// TwinCAT 3 PLC project MicroTestStandWFS
// ProgramVersion: 3.1.4020.5
// libraries:
//   lcls-twincat-motion, * (SLAC)
//   lcls2-cc-lib, * (SLAC)
//   PMPS, * (SLAC - LCLS)
//   Tc2_Standard, * (Beckhoff Automation GmbH)
//   Tc2_System, * (Beckhoff Automation GmbH)
//   Tc2_Utilities, * (Beckhoff Automation GmbH)
//   Tc3_Module, * (Beckhoff Automation GmbH)
//   VisuDialogs
//   VisuSymbols,3.5.10.0,System
// project tree:
//   DUTs/ DUT_MotionStage_Extras.TcDUT (not stored)
//   / GlobalTextList.TcGTLO, PlcTask.TcTTO (not stored), VISU_TASK.TcTTO (not stored)
//   POUs/ Main.TcPOU
//   VISUs/ Visualization.TcVIS, VisualizationManager.TcVMO (not stored), VISU_MotionStage.TcVIS (not stored)

// ---- POUs/Main.TcPOU
PROGRAM Main
VAR
	{attribute 'TcLinkTo' := '.bLimitForwardEnable  := TIIB[EL7041-Y]^STM Status^Status^Digital input 1;
	                          .bLimitBackwardEnable := TIIB[EL7041-Y]^STM Status^Status^Digital input 2;
	                          .bBrakeRelease        := TIIB[EL2004]^Channel 1^Output'}
	M1: DUT_MotionStage;
	M1_Extras: DUT_MotionStage_Extras;
    
	M2: DUT_MotionStage;
	M2_Extras: DUT_MotionStage_Extras;
	
	{attribute 'TcLinkTo' := '.fbThermoCouple1.bError := TIIB[EL3314]^TC Inputs Channel 1^Status^Error;
							  .fbThermoCouple1.bUnderrange := TIIB[EL3314]^TC Inputs Channel 1^Status^Underrange;
							  .fbThermoCouple1.bOverrange := TIIB[EL3314]^TC Inputs Channel 1^Status^Overrange;
							  .fbThermoCouple1.iRaw := TIIB[EL3314]^TC Inputs Channel 1^Value;
							  .fbThermoCouple2.bError := TIIB[EL3314]^TC Inputs Channel 2^Status^Error;
							  .fbThermoCouple2.bUnderrange := TIIB[EL3314]^TC Inputs Channel 2^Status^Underrange;
							  .fbThermoCouple2.bOverrange := TIIB[EL3314]^TC Inputs Channel 2^Status^Overrange;
							  .fbThermoCouple2.iRaw := TIIB[EL3314]^TC Inputs Channel 2^Value'}
	fbWFS: FB_WFS;
	

    {attribute 'TcLinkTo' := 'TIIB[EL5042]^FB Inputs Channel 2^Position'}
	iM1RawEncoder AT %I*: ULINT;
	iM1AdjustedEncoder: UDINT;
    
    {attribute 'TcLinkTo' := 'TIIB[EL5042]^FB Inputs Channel 1^Position'}
    iM2RawEncoder AT %I*: ULINT;
    iM2AdjustedEncoder: UDINT;
    
	iMaxLINT: ULINT := 18446744073709551615;
	
	bStartup: BOOL := TRUE;
    
    // PMPS Machinery
    fbArbiterIO: FB_SubSysToArbiter_IO;
    {attribute 'pytmc' := 'pv: PLC:TST:MOT:ARB'}
    fbArbiter: FB_Arbiter(1);
    {attribute 'pytmc' := 'pv: PLC:TST:MOT:FFO:01'}
    fbFFHWO: FB_HardwareFFOutput := (bAutoReset := TRUE);
END_VAR

fbWFS(
    stYStage := M1,
    stZStage := M2,
    fbArbiter := fbArbiter,
    fbFFHWO:=fbFFHWO);

fbFFHWO.Execute();
fbArbiterIO(
    Arbiter:=fbArbiter,
    fbFFHWO:=fbFFHWO);


iM1AdjustedEncoder := ULINT_TO_UDINT(iMaxLINT - iM1RawEncoder) + 1;
iM2AdjustedEncoder := ULINT_TO_UDINT(iM2RawEncoder);

M1_Extras.bVisuHighLim := NOT M1.bAllForwardEnable;
M1_Extras.bVisuLowLim := NOT M1.bAllBackwardEnable;
M2_Extras.bVisuHighLim := NOT M2.bAllForwardEnable;
M2_Extras.bVisuLowLim := NOT M2.bAllBackwardEnable;

IF bStartup THEN
	bStartup := FALSE;
	M1.fVelocity := 1;
	M1.fAcceleration := 200;
	M1.fDeceleration := 200;
	M2.fVelocity := 1;
	M2.fAcceleration := 200;
	M2.fDeceleration := 200;
END_IF

END_PROGRAM

// ---- GlobalTextList.TcGTLO
TEXTLIST GlobalTextList
  593 = '%f'
  964 = '%X'
  957 = '+'
  951 = '-'
  960 = '0 = Default Acceleration'
  962 = '0 = Default Deceleration'
  959 = 'Acceleration: %f'
  504 = 'Cam Power'
  955 = 'Clear'
  582 = 'Close Screen'
  949 = 'Control'
  684 = 'Controls'
  594 = 'Current Position'
  961 = 'Deceleration: %f'
  324 = 'Encoder'
  965 = 'Error Code'
  963 = 'Error:'
  953 = 'GO'
  954 = 'GO to set position'
  595 = 'High Limit Hit Indicator'
  768 = 'Illuminator: %f %'
  592 = 'Low Limit Hit Indicator'
  30 = 'Motion Stage'
  460 = 'Motor'
  596 = 'Moving:'
  311 = 'Parker Stage'
  109 = 'PM TC: %f C'
  658 = 'PM Temp: %f C'
  598 = 'Power Meter: %f V'
  921 = 'PPM'
  890 = 'Raw count: %d'
  7 = 'Raw count: %f'
  274 = 'Readbacks'
  950 = 'Set Position'
  470 = 'Settings'
  591 = 'Status'
  952 = 'Step Size'
  956 = 'STOP'
  917 = 'Temp 1: %f C'
  256 = 'Temp 2: %f C'
  151 = 'Thermocouple Readbacks'
  958 = 'Velocity: %f'
  562 = 'X Motor'
  568 = 'Y Motor'
  316 = 'Yag Temp: %f C'
  824 = 'Z Motor'
END_TEXTLIST

// ---- VISUs/Visualization.TcVIS
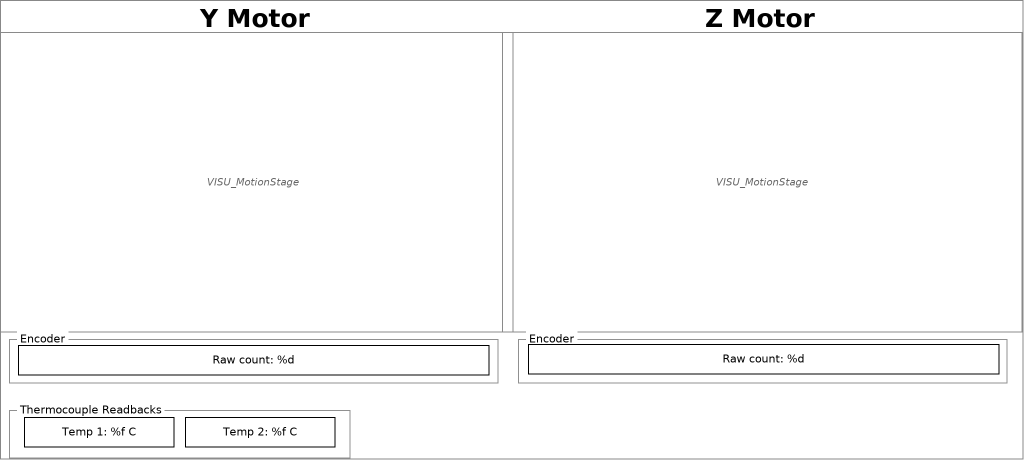
VISUALIZATION Visualization  // 1024x460
    Label (14,3 482x30), "Y Motor"
    Label (519,3 482x30), "Z Motor"
    GroupBox (9,402 341x56), "Thermocouple Readbacks"
        Rectangle (15,15 150x30), "Temp 1: %f C", text variable: Main.fbWFS.fbThermoCouple1.fTemp
        Rectangle (176,15 150x30), "Temp 2: %f C", text variable: Main.fbWFS.fbThermoCouple2.fTemp
    Frame (-7,32 520x300)
        shows VISU_MotionStage(VisuMotionStage := Main.M1, Extras := Main.M1_Extras)
    Frame (502,32 520x300)
        shows VISU_MotionStage(VisuMotionStage := Main.M2, Extras := Main.M2_Extras)
    GroupBox (9,331 489x52), "Encoder"
        Rectangle (9,14 471x30), "Raw count: %d", text variable: Main.iM1AdjustedEncoder
    GroupBox (518,331 489x52), "Encoder"
        Rectangle (10,13 471x30), "Raw count: %d", text variable: Main.iM2AdjustedEncoder
END_VISUALIZATION
